INTERFACE I_PositioningHomingBuilder EXTENDS __System.IQueryInterface

METHOD BuildDefaultHomingCommand : I_HomingCommand
END_METHOD

METHOD BuildDirectHomingCommand : I_HomingCommand
END_METHOD

METHOD Cam : I_DefaultHomingBuilder
VAR_INPUT
	value : REFERENCE TO BOOL;
END_VAR
END_METHOD

METHOD ClearLag : I_PositioningHomingBuilder
END_METHOD

METHOD KeepLag : I_PositioningHomingBuilder
END_METHOD

METHOD Position : I_PositioningHomingBuilder
VAR_INPUT
	value : LREAL;
END_VAR
END_METHOD

METHOD ReferenceMode : I_DefaultHomingBuilder
VAR_INPUT
	value : EncoderReferenceMode;
END_VAR
END_METHOD

METHOD SearchDirection : I_DefaultHomingBuilder
VAR_INPUT
	value : Direction;
END_VAR
END_METHOD

METHOD SearchVelocity : I_DefaultHomingBuilder
VAR_INPUT
	value : LREAL;
END_VAR
END_METHOD

METHOD SyncDirection : I_DefaultHomingBuilder
VAR_INPUT
	value : Direction;
END_VAR
END_METHOD

METHOD SyncVelocity : I_DefaultHomingBuilder
VAR_INPUT
	value : LREAL;
END_VAR
END_METHOD

END_INTERFACE

(* stored: Version 1.1.0.1, ProductVersion 3.1.4024.12
   Itf I_PositioningHomingBuilder: Id {b83c6e00-d80a-4eee-9c0a-7bfcc12039a8}
   Method BuildDefaultHomingCommand: Id {0443752a-d7ca-446b-8596-fb433e8cb64d}
   Method BuildDirectHomingCommand: Id {40713a8c-4ea3-48b9-aac6-b2db3d62d563}
   Method Cam: Id {06b8b962-bd76-402f-83e8-d05a099573f9}
   Method ClearLag: Id {866850ba-07ba-46bf-b37a-f8110351fe16}
   Method KeepLag: Id {424b73d3-98f6-41ea-a5c1-72797f933ac5}
   Method Position: Id {53bbd10d-edd8-4df6-b098-33c26980dd34}
   Method ReferenceMode: Id {937aeae7-2045-4249-b725-e6501ef3ab37}
   Method SearchDirection: Id {a7938a16-e3a7-4cc7-9980-8edc187a8ed3}
   Method SearchVelocity: Id {22c99f85-2366-44c9-ba7a-12f2598873f9}
   Method SyncDirection: Id {d65a817d-257f-4de6-a581-cd3725ce701a}
   Method SyncVelocity: Id {9e7b4817-7fc5-4c4b-856f-11c8ead0e230} *)
